{attribute 'qualified_only'}
TYPE PAOperatingModeEnum :
(
	Automatic := 0,
	Manual := 1,
	Maintenance := 2
);
END_TYPE

(* stored: Version 1.1.0.1, ProductVersion 3.1.4020.12
   DUT PAOperatingModeEnum: Id {d6291495-38df-4718-919e-2d649f2037ab} *)
